FUNCTION_BLOCK FB_HeavyWash IMPLEMENTS I_WashStrategy
VAR
	 bStarted : BOOL := FALSE; 
	 stSettings : ST_WashSettings;
END_VAR

METHOD FB_init : BOOL
VAR_INPUT
	bInitRetains : BOOL; // if TRUE, the retain variables are initialized (warm start / cold start)
	bInCopyCode : BOOL;  // if TRUE, the instance afterwards gets moved into the copy code (online change)
END_VAR
stSettings.rTemperature  := GVL_WashConstants.HEAVY_TEMP; 
stSettings.nSpinSpeed    := GVL_WashConstants.HEAVY_SPIN; 
stSettings.tWashDuration := GVL_WashConstants.HEAVY_WASH_TIME; 
stSettings.sDescription  := GVL_WashConstants.HEAVY_DESC; 

FB_init := TRUE;
END_METHOD

METHOD GetDuration : TIME
GetDuration := stSettings.tWashDuration ;
END_METHOD

METHOD GetProgramName : STRING
GetProgramName := 'HEAVY';
END_METHOD

METHOD GetSettings : ST_WashSettings
GetSettings := stSettings;
END_METHOD

METHOD Start : BOOL
bStarted := TRUE; 
Start     := TRUE;
END_METHOD

END_FUNCTION_BLOCK

(* stored: Version 1.1.0.1, ProductVersion 3.1.4024.16
   POU FB_HeavyWash: Id {b328f795-7fca-4f9b-befa-cc3fc249bc0e}, SpecialFunc None
   Method FB_init: Id {6bba0abe-2e8b-4730-ae6a-c44784daf780}
   Method GetDuration: Id {86db14ab-625b-4bb7-a994-003ec6a66b96}
   Method GetProgramName: Id {8637de0d-40fd-42ba-804e-ccf96594f716}
   Method GetSettings: Id {48daccf0-d622-4f0c-8fd4-c7412b99fd2e}
   Method Start: Id {78e9b4e5-1a49-435d-995b-4ef35591c35a} *)
